PROGRAM TESTS
VAR
//	Test_Extend_TurnsOnValve_And_ReportsExtended 	: FB_Cylinder_Test;
//	Test_MockedExecutor 							: FB_ExecutorCut_Test; 
//	Test_ExecutorGCode  							: FB_ExecutorGCode_Test;
//	Test_GrooveExecutor 							: FB_ExecutorGrooveXY_Test;
//	Test_ExecutorNCITable							: FB_ExecutorNCITable_Test;
//	Test_FeedBuilderRoundedRect 					: FB_FeedBuilderRoundedRect_Test;
//	Test_GantryXYZ									: FB_GantryXYZ_Test;
//	Test_NciChannel            						: FB_NciChannel_Test;
//  Test_NciChannelTangential  						: FB_NciChannelTangential_Test; // Mock Channel
//	Test_RecipeBuilder 								: FB_RecipeBuilder_Test;
//	Test_RecipeFactory 								: FB_RecipeFactory_Test;
//	Test_FB_Exec_Drill_PTP_Test						: FB_Exec_Drill_PTP_Test;
END_VAR

//TcUnit.RUN();

END_PROGRAM

(* stored: Version 1.1.0.1, ProductVersion 3.1.4024.15
   POU TESTS: Id {0938b2ab-3336-43f1-a2aa-780b5d2a82ee}, SpecialFunc None *)
